{attribute 'Tc2GvlVarNames'}
{attribute 'strict'}
//Stato della lista DI PRODUZIONE
TYPE e_Stato_ListaDiProduzione :
(
	LISTA_PROD_NOT_DEFINED 		:= -1, 	//STATO LISTA PRODODUZIONE NON DEFINITO
	LISTA_PROD_ASSENTE			:= 0,	//STATO LISTA PRODODUZIONE ASSENTE:	In questo caso la macchina su questa Postazione non effettuerà alcuna lavorazione di deposito "Per composizione"
	LISTA_PROD_DA_ESEGUIRE 		:= 1, 	//STATO LISTA PRODODUZIONE DA ESEGUIRE
	LISTA_PROD_IN_ESECUZIONE 	:= 2,	//STATO LISTA PRODODUZIONE IN ESECUZIONE
	LISTA_PROD_ESEGUITA 		:= 3	//STATO LISTA PRODODUZIONE ESEGUITA
);
END_TYPE
//  LISTA_PROD_NOT_DEFINED = '-1'

(* stored: Version 1.1.0.1, ProductVersion 3.1.4024.11
   EnumerationTextList e_Stato_ListaDiProduzione: Id {8d29cca0-d483-402a-a44b-24a139f3ca5d} *)
